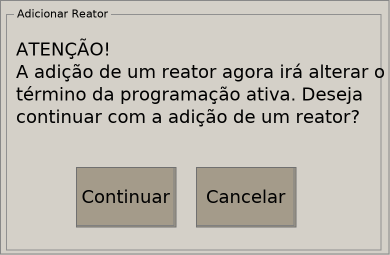
VISUALIZATION Notifica24horas  // 390x255
    GroupBox (6,6 375x244), "Adicionar Reator"
        Label (7,31 373x126), "ATENÇÃO! A adição de um reator agora irá alterar o término da programação ativa. Deseja continuar com a adição de um reator?"
        Button (70,161 100x60), "Continuar"
            OnMouseClick: execute {
                posCarrinho.bNotificaTime:=TRUE;
                posCarrinho2.bNotificaTime:=TRUE;
                posCarrinho3.bNotificaTime:=TRUE;
            }
        Button (190,161 100x60), "Cancelar"
            OnMouseClick: CloseDialog Dialog=ConfigPosicao_Reator, Result=Cancel, NumpadKeypadSet=True
            OnMouseClick: execute {
                posCarrinho.bNotificaTime:=TRUE;
                posCarrinho2.bNotificaTime:=TRUE;
                posCarrinho3.bNotificaTime:=TRUE;
            }
            OnMouseClick: CloseDialog Dialog=ConfigPosicao_Reator_2, Result=Cancel, NumpadKeypadSet=True
            OnMouseClick: CloseDialog Dialog=ConfigPosicao_Reator_3, Result=Cancel, NumpadKeypadSet=True
END_VISUALIZATION

(* stored: Version 1.1.0.1, ProductVersion 3.1.4024.12
   Visu Notifica24horas: Id {072b6c79-c064-4d14-a612-fe545f15e8a0} *)
